TYPE ST_SettingsAirTrearment :
STRUCT
	fPressurizingPress : LREAL; //[Pa]
	fFlushingPress : LREAL; //[Pa]
	tFlushingTime : TIME; //[s]
	fEqualizingPress : LREAL; //[Pa]
	fRange : LREAL; //[Pa]
	fKp : LREAL; //Proportional gain Kp (P)
    fTn : LREAL; //Integral gain Tn (I) [s]
    fTv : LREAL; //Derivative gain Tv (D-T1) [s]
    fTd : LREAL; //Derivative damping time Td (D-T1) [s]
END_STRUCT
END_TYPE

(* stored: Version 1.1.0.1, ProductVersion 3.1.4024.12
   DUT ST_SettingsAirTrearment: Id {06fc4816-030f-4763-8a01-113573740184} *)
